PROGRAM gesAlarmas
VAR
	TempTimeOUT:ton;
	EstAnt:EstadosPrensa;
	
	PrimeiroErro:INT;
	Erros:ARRAY[1..9] OF BOOL;
	contador:INT;

END_VAR

IF Variablesglobales.ModoMaquina=modos.Reseteando THEN
	primeiroerro:=0;
	FOR contador:=1 TO 9 DO
		erros[contador]:=FALSE;
	END_FOR
END_IF

temptimeout(in:=estant=modoautomatico.EstadoPrensa AND 
	variablesglobales.ModoMaquina = modos.Auto AND 
	modoautomatico.estadoprensa <> estadosprensa.Parada, pt:=T#15S); //la vaina esta <> es un distinto
IF tempTimeout.q THEN 
	erros[1]:=TRUE;
	IF primeiroErro=0 THEN
		primeiroErro:=1;
	END_IF
END_IF

//error ejes
IF ErrorEjes THEN
	erros[2]:=TRUE;
	IF primeiroerro=0 THEN
		primeiroerro:=2;
	END_IF
END_IF

//seta emergency
IF NOT io.SafetyOK THEN
	erros[3]:=TRUE;
	IF primeiroerro=0 THEN
		primeiroerro:=3;
	END_IF	
END_IF

//mando dos manos
IF mandoa2mans.Error THEN
	erros[4]:=TRUE;
	IF primeiroerro=0 THEN
		primeiroerro:=4;
	END_IF	
END_IF

VariablesGlobales.EnErro := PrimeiroErro<>0;
estant:=modoautomatico.EstadoPrensa;

END_PROGRAM

(* stored: Version 1.1.0.1, ProductVersion 3.1.4024.9
   POU gesAlarmas: Id {197760f4-3c71-4d0b-adc6-89bfdb36f692}, SpecialFunc None *)
